Yaskawa INFORM job: R2_W68-69(-90,-90)AWOK.JBI

/JOB
//NAME R2_W68-69(-90,-90)AWOK
///FOLDERNAME AWOK
//POS
///NPOS 40,40,0,3,0,0
///TOOL 0
///POSTYPE PULSE
///PULSE
C00000=73468,9895,-28016,-5981,91523,26793
C00001=120734,71276,72201,4504,87810,-53709
C00002=120735,71272,72196,4504,87811,-53709
C00003=120735,71272,72196,4504,87811,-53709
C00004=120735,71697,73169,4504,87433,-53721
C00005=120735,71270,72194,4504,87811,-53709
C00006=120735,71182,72087,15370,72811,-50996
C00007=120779,71193,72101,15365,72800,-50982
C00008=120735,71182,72087,15370,72811,-50996
C00009=120735,71325,72260,-1559,94818,-55545
C00010=120735,69399,69950,-1560,95249,-55550
C00011=120735,71325,72260,-1559,94818,-55545
C00012=120735,71328,72263,-1559,94817,-55545
C00013=120734,71336,72273,-1559,94815,-55545
C00014=120751,61561,41578,27514,97921,23508
C00015=120734,70951,71810,-2171,75229,66298
C00016=120734,70920,71772,-2171,75236,66298
C00017=120735,70907,71757,-2171,75239,66298
C00018=120735,71396,72877,-2175,74802,66306
C00019=120735,70907,71757,-2171,75239,66298
C00020=120735,70960,71820,-8595,68252,65467
C00021=120735,69136,69634,-8572,68656,65436
C00022=120735,70960,71820,-8595,68252,65467
C00023=120735,70816,71648,4347,82003,67463
C00024=120500,70806,71637,4342,82017,67384
C00025=120735,70816,71648,4347,82003,67463
C00026=120734,70827,71660,4347,82001,67463
C00027=120734,70853,71692,4347,81995,67463
C00028=112400,61296,37228,-23103,109629,-28450
C00029=107341,71278,72203,-37113,101922,-81721
C00030=107341,71251,72171,-37114,101927,-81723
C00031=84559,41524,23043,1779,100366,-86516
C00032=107467,74944,76649,-36953,101288,-81446
C00033=107434,72961,73317,-37117,102107,-81746
C00034=112989,15210,-1991,9801,101125,-76428
C00035=112598,15517,-77,16334,100667,-76359
C00036=109663,20975,-134,16743,105523,-76722
C00037=109663,20975,-134,16743,105523,-76722
C00038=109630,25453,-16548,18427,117386,-74878
C00039=-3792,5914,-36214,18652,-1261,-74575
BC00000=44418,319272,865261
BC00001=87328,212950,591893
BC00002=84135,215207,568566
BC00003=82858,216109,559235
BC00004=82874,216111,551757
BC00005=82858,216109,559235
BC00006=99536,246297,551426
BC00007=97147,246299,551369
BC00008=99536,246297,551426
BC00009=70662,206515,552384
BC00010=70663,208370,552391
BC00011=70662,206515,552384
BC00012=71596,205193,561564
BC00013=73933,201888,584513
BC00014=161167,225184,507004
BC00015=155724,234952,604802
BC00016=157686,236656,579439
BC00017=158471,237338,569294
BC00018=158488,237340,561229
BC00019=158471,237338,569294
BC00020=146517,255975,562174
BC00021=146538,258072,562182
BC00022=146517,255975,562174
BC00023=176585,221848,566781
BC00024=178974,221826,566838
BC00025=176585,221848,566781
BC00026=176188,220784,576780
BC00027=175193,218125,601776
BC00028=108792,188298,523388
BC00029=68701,170289,476059
BC00030=71515,176017,460875
BC00031=72469,177959,455726
BC00032=72640,178308,454802
BC00033=72640,178308,454802
BC00034=72469,177959,455727
BC00035=72469,177959,455727
BC00036=72469,177959,455727
BC00037=72469,177959,455727
BC00038=72469,177958,455723
BC00039=72469,294340,455723
///POSTYPE BASE
///RECTAN
///RCONF 0,0,0,0,0,0,0,0,0,0,0,0,0,0,0,0,0,0,0,0,0,0,0,0
P00006=0.222,-3.123,-1.508,0.0000,0.0000,0.0000
P00021=-0.225,-6.128,-0.405,0.0000,0.0000,0.0000
P00022=0.222,-3.123,-1.508,0.0000,0.0000,0.0000
//INST
///DATE 2023/11/16 10:49
///ATTR SC,RW
///GROUP1 RB1,BS1
NOP
'OK ALE SEARCH MOZNA OPTYM
'r2_W68-69(-90,-90)
'Path S758 (for W102)
SFTOF
MOVJ C00000 BC00000 VJ=20.00
MOVJ C00001 BC00001 VJ=20.00
MOVL C00002 BC00002 V=100.0
MOVL C00003 BC00003 V=60.0
REFP 3 C00004 BC00004
CALL JOB:SEARCH-R1
SET P021 P006
SFTON P021
MOVL C00005 BC00005 V=60.0
MOVL C00006 BC00006 V=60.0
REFP 3 C00007 BC00007
CALL JOB:SEARCH-R1
SET P021 P006
SFTON P021
MOVL C00008 BC00008 V=60.0
MOVL C00009 BC00009 V=60.0
REFP 3 C00010 BC00010
CALL JOB:SEARCH-R1
SET P021 P006
SFTON P021
MOVL C00011 BC00011 V=60.0
MOVL C00012 BC00012 V=100.0
MOVL C00013 BC00013 V=100.0
'Path VIA1138
SFTOF
MOVJ C00014 BC00014 VJ=20.00
'Path S759 (for W102)
SFTOF
MOVJ C00015 BC00015 VJ=20.00
MOVL C00016 BC00016 V=100.0
MOVL C00017 BC00017 V=60.0
REFP 3 C00018 BC00018
CALL JOB:SEARCH-R1
SET P022 P006
SFTON P022
MOVL C00019 BC00019 V=60.0
MOVL C00020 BC00020 V=60.0
REFP 3 C00021 BC00021
CALL JOB:SEARCH-R1
SET P022 P006
SFTON P022
MOVL C00022 BC00022 V=60.0
MOVL C00023 BC00023 V=60.0
REFP 3 C00024 BC00024
CALL JOB:SEARCH-R1
SET P022 P006
SFTON P022
MOVL C00025 BC00025 V=60.0
MOVL C00026 BC00026 V=100.0
MOVL C00027 BC00027 V=100.0
'Path VIA1139
SFTOF
MOVJ C00028 BC00028 VJ=20.00
'Path W102
SFTOF
SFTON P022
MOVJ C00029 BC00029 VJ=20.00
MOVL C00030 BC00030 V=100.0
MOVL C00031 BC00031 V=100.0 PL=0
REFP 1 C00032 BC00032
REFP 2 C00033 BC00033
MACRO1 MJ#(0) ARGF9
ARCON
SFTON P021
MOVL C00034 BC00034 V=10.8
MOVL C00035 BC00035 V=10.8
ARCOF
MOVL C00036 BC00036 V=100.0
MOVL C00037 BC00037 V=100.0
SFTOF
MOVJ C00038 BC00038 VJ=20.00
MOVJ C00039 BC00039 VJ=20.00
END
